FUNCTION_BLOCK INIT_ARR_007_BYTE (* FB to make an Array *)
  (* Standard: 61499-2 *)
  (* Version 1.0, 2026-01-22, Franz Höpfinger, Andreas Demmler Fahrzeugbau *)
  PACKAGE logiBUS::utils::generate;
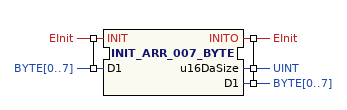
  EVENT_INPUT
    INIT : EInit WITH D1; (* Service Initialization *)
  END_EVENT
  EVENT_OUTPUT
    INITO : EInit WITH u16DaSize, D1; (* Initialization Confirm *)
  END_EVENT
  VAR_OUTPUT
    u16DaSize : UINT; (* Data length in Array Elements *)
  END_VAR
  VAR_IN_OUT
    D1 : ARRAY [0..7] OF BYTE; (* Data *)
  END_VAR
END_FUNCTION_BLOCK
